// Mitsubishi GX Works2 project: 一些输出的有意思方法   PLC: Q13UDV

TYPE movdate : STRUCT
  inout : ;
END_STRUCT END_TYPE

FUNCTION_BLOCK mov_out
VAR_OUTPUT
  date_out : INT;
END_VAR
VAR_INPUT
  气缸下降破真空 : BOOL;  (* 气缸下降破真空 *)
  气缸下降吸真空 : BOOL;  (* 气缸下降吸真空 *)
  气缸上升破真空 : BOOL;  (* 气缸上升破真空 *)
  气缸上降吸真空 : BOOL;  (* 气缸上降吸真空 *)
END_VAR
IF 
气缸下降破真空
 THEN date_out
:= 2#1001;
     ELSE IF 气缸下降吸真空 THEN date_out
 := 2#0101;
     ELSE IF 气缸上升破真空 THEN date_out
 := 2#1010;
     ELSE IF 气缸上降吸真空 THEN date_out
:= 2#0110;
     ELSE date_out
 := 0;   
END_IF;END_IF;END_IF;END_IF;





D0:=D0+k1;
END_FUNCTION_BLOCK

PROGRAM inout
VAR
  气缸下降真空打开 : mov_out;
END_VAR
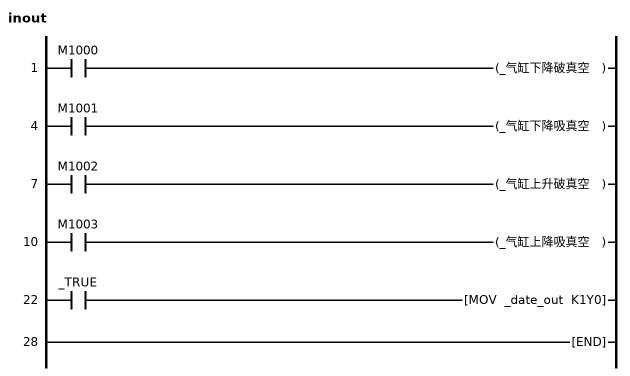
; FB BLK START mov_out(气缸下降真空打开)
1     LD      M1000
      OUT     _气缸下降破真空
4     LD      M1001
      OUT     _气缸下降吸真空
7     LD      M1002
      OUT     _气缸上升破真空
10    LD      M1003
      OUT     _气缸上降吸真空
; FB START
; FB_NAME mov_out
; INSTANCE_NAME 气缸下降真空打开
; FB IN_B:气缸下降破真空
; FB OUT_date_out:W
; FB IN_B:气缸下降吸真空
; FB IN_B:气缸上升破真空
; FB IN_B:气缸上降吸真空
; FB END
22    LD      _TRUE
      MOV     _date_out K1Y0  ; 下降气缸
; FB BLK END
28    END
END_PROGRAM

// device comments not shown above
Y1  ; 上升气缸
Y2  ; 真空气缸
Y3  ; 破真空气缸
Y4  ; 旋转气缸
